(* FB_CylinderDiag	- number of control signals:
							one direction is controllable
					- type of feedback signal:
							feedback in base and work position
					- with position diagnosis						*)
					
FUNCTION_BLOCK FB_CylinderDiag EXTENDS FB_Cylinder
VAR_INPUT
	tTimeOut 	 		: TIME;			// Time for watchdog that monitores if cylinder reaches base/work position
END_VAR
VAR_OUTPUT
	bError				: BOOL;			// Error signal (diagnosed from position watchdog)
	sErrorMsg			: STRING;		// Error message
END_VAR
VAR
	fbTriggerError		: R_TRIG;		// Trigger to recognize rising edge of error
	bErrorMove			: BOOL;			// Move error
	fbTimerWatchDog		: TON;			// Watchdog timer for monitoring if cylinder reaches base/work position
END_VAR

// =========================================================
;
// =========================================================

METHOD PROTECTED Diag
VAR_INPUT
END_VAR
// =========================================================
// Timer starts when cylinder is not in base and work position
	
	IF NOT bAtBasePos AND NOT bAtWorkPos THEN
		fbTimerWatchDog(IN := TRUE,
						PT := tTimeOut);
	ELSE
		fbTimerWatchDog(IN := FALSE,
						PT := tTimeOut);
	END_IF

// =========================================================
// Error if cylinder does not reach base or work position
	
	fbTriggerError(CLK := fbTimerWatchDog.Q);
	
	bError := fbTimerWatchDog.Q;
	
	IF fbTriggerError.Q THEN
		bErrorMove := bMoveToWork;
	END_IF
	
	IF bError THEN
		IF bErrorMove = bMoveToWork THEN
			IF bMoveToWork THEN
				sErrorMsg := 'Work position not reached';
			ELSE
				sErrorMsg := 'Base position not reached';
			END_IF
		ELSE
			bError := FALSE;
			sErrorMsg := '';
		END_IF
	ELSE
		sErrorMsg := '';
	END_IF

// =========================================================
END_METHOD

METHOD Reset
VAR_INPUT
END_VAR
// =========================================================

// Calling method Reset of base class FB_Cylinder via 'SUPER^.'
SUPER^.Reset();		

// Reset error
bError 		:= FALSE;
sErrorMsg 	:= '';

// =========================================================
END_METHOD

METHOD PROTECTED StateMachine
VAR_INPUT
	bBasePosReq		: BOOL;
	bWorkPosReq		: BOOL;
END_VAR
// =========================================================

IF NOT bError THEN
	// Calling method StateMachine of base class FB_Cylinder via 'SUPER^.'
	SUPER^.StateMachine(bBasePosReq := bBasePosReq,
						bWorkPosReq	:= bWorkPosReq );
	
	// Diagnosis
	Diag();
END_IF

// =========================================================
END_METHOD

END_FUNCTION_BLOCK

(* stored: Version 1.1.0.1, ProductVersion 3.1.4024.12
   POU FB_CylinderDiag: Id {b98e6e0a-c06c-4bfd-9411-67daeb0dbabb}, SpecialFunc None
   Method Diag: Id {f79f365d-dffb-4a7d-9fa6-75d28cecb63b}
   Method Reset: Id {4201fe92-72e6-40bb-ba50-b855cb4acd15}
   Method StateMachine: Id {28ea0f6a-96f6-4957-90a0-49a2f6f68a26} *)
